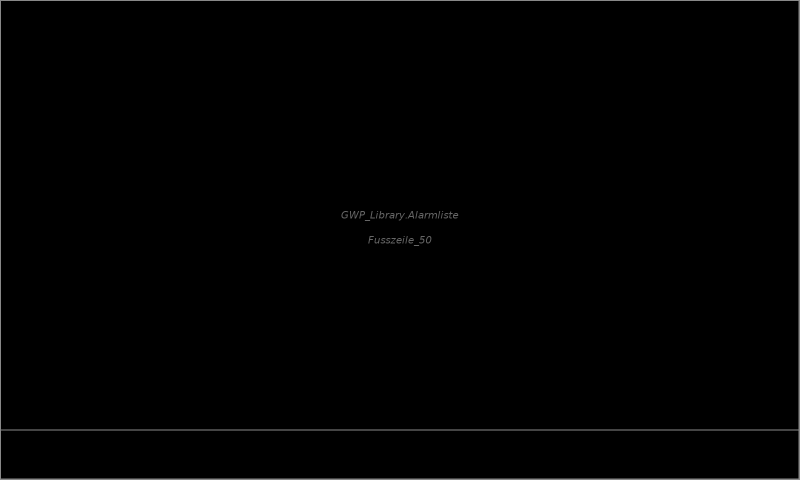
VISUALIZATION Alarmliste  // 800x480
    Frame (0,0 800x480)
        shows Fusszeile_50()
    Frame (0,0 800x430)
        shows GWP_Library.Alarmliste()
END_VISUALIZATION

(* stored: Version 1.1.0.1, ProductVersion 3.1.4022.6
   Visu Alarmliste: Id {ea16c1c0-4094-48f6-bbb7-037f4fe26be9} *)
